(* CODESYS project HomePLC_DIO.library
   Company: Tom Oyen
   Description: Digital in- and outputs
   Version: 1.0
   Placeholder: HomePLC DIO
   Author: Tom Oyen
   Title: HomePLC DIO

Project tree, tasks and I/O mapping:
  libraries: HomePLC Logging, * (Tom Oyen); Tc2_Standard, * (Beckhoff Automation GmbH); Tc2_System, * (Beckhoff Automation GmbH); Tc3_Module, * (Beckhoff Automation GmbH)
  POUs/
    DI/
      DUTs/
        data type E_DICommand
        data type E_DIExecuteSteps
        data type E_DIState
        data type ST_HmiDigitalIn
      function block FB_DigitalIn [ST]: EnableDefer, EnableDoublePress, Execute, SetExternalIn, Command, HmiData, State
      interface I_DigitalIn: EnableDefer, EnableDoublePress, SetExternalIn, Command, HmiData, State
    DO/
      DUTs/
        data type E_DOCommand
        data type E_DOFlashStep
        data type E_DOState
        data type ST_HmiDigitalOut
      function block FB_DigitalOut [ST]: Execute, SetBlinkPeriod, SetCommand, SetFlashTime, BlinkPeriod, Command, FlashTime, HmiData, State
      function block FB_SquareWave [ST]
      interface I_DigitalOut: SetBlinkPeriod, SetCommand, SetFlashTime, BlinkPeriod, Command, FlashTime, HmiData, State
    function block FB_DIO [ST]: Execute, FB_init, Name
    interface I_DIO: Execute, Name
  Project Information/
    function F_GetCompany [ST]
    function F_GetTitle [ST]
    function F_GetVersion [ST]
  Version/
    global variables Global_Version
*)

// POUs/DI/DUTs/E_DICommand
{attribute 'qualified_only'}
{attribute 'strict'}
{attribute 'to_string'}
// Digital input command (generated by digital input)
TYPE E_DICommand :
(
	None		:= 0,		// No input action
	ShortPress	:= 1,		// Input pressed for short amount of time
	LongPress	:= 2,		// Input pressed for longer amount of time but not held
	DoublePress	:= 3,		// Input double pressed
	Hold		:= 4		// Input held for long amount of time
);
END_TYPE

// POUs/DI/DUTs/E_DIExecuteSteps
{attribute 'qualified_only'}
{attribute 'strict'}
// Digital input state machine steps
TYPE E_DIExecuteSteps :
(
	Idle					:= 0,
	FirstShortPressDetected	:= 1,
	WaitForSecondPress		:= 2,
	ShortPressDetected		:= 3,
	DoublePressDetected		:= 4,
	LongPressDetected		:= 5,
	HoldDetected			:= 6,
	WaitUntilReleased		:= 7,
	Reset					:= 8
);
END_TYPE

// POUs/DI/DUTs/E_DIState
{attribute 'qualified_only'}
{attribute 'strict'}
{attribute 'to_string'}
// Digital input state
TYPE E_DIState :
(
	Idle			:= 0,		// No input action
	Pressing1		:= 1,		// Input is being pressed for the first time for a short amount of time
	LongPressing	:= 2,		// Input is being pressed longer
	Pressing2		:= 3,		// Input is being pressed for the second time
	Holding			:= 4,		// Input is being held
	Deferring		:= 5
);
END_TYPE

// POUs/DI/DUTs/ST_HmiDigitalIn
TYPE ST_HmiDigitalIn :
STRUCT
	sName	: STRING;
	eState	: E_DIState;
	bValue	: BOOL;
END_STRUCT
END_TYPE

// POUs/DO/DUTs/E_DOCommand
{attribute 'qualified_only'}
{attribute 'strict'}
{attribute 'to_string'}
// Digital output command (received by digital output)
TYPE E_DOCommand :
(
	None		:= 0,		// No command given
	On			:= 1,		// Turn on
	Off			:= 2,		// Turn off
	Toggle		:= 3,		// Toggle
	Blink		:= 4,		// Blink continuously
	Flash		:= 5		// Flash once (either flash on when already off or flash off when already on)
);
END_TYPE

// POUs/DO/DUTs/E_DOFlashStep
{attribute 'qualified_only'}
{attribute 'strict'}
// Steps when flashing
TYPE E_DOFlashStep :
(
	Start					:= 0,
	ToggleOutput			:= 1,
	WaitForTimer			:= 2,
	RestoreOutput			:= 3,
	End						:= 4
);
END_TYPE

// POUs/DO/DUTs/E_DOState
{attribute 'qualified_only'}
{attribute 'strict'}
{attribute 'to_string'}
// Digital output state
TYPE E_DOState :
(
	Idle			:= 0,		// Idle
	TurnOn			:= 1,		// Turn on
	TurnOff			:= 2,		// Turn off
	Toggle			:= 3,		// Toggle
	Blinking		:= 4,		// Blinking
	Flashing		:= 5		// Flashing	
);
END_TYPE

// POUs/DO/DUTs/ST_HmiDigitalOut
TYPE ST_HmiDigitalOut :
STRUCT
	sName	: STRING;
	eState	: E_DOState;
	bValue	: BOOL;
END_STRUCT
END_TYPE

// Version/Global_Version
{attribute 'TcGenerated'}
{attribute 'no-analysis'}
{attribute 'linkalways'}
// This function has been automatically generated from the project information.
VAR_GLOBAL CONSTANT
	{attribute 'const_non_replaced'}
	stLibVersion_HomePLC_DIO : ST_LibVersion := (iMajor := 1, iMinor := 0, iBuild := 0, iRevision := 0, nFlags := 0, sVersion := '1.0');
END_VAR

// POUs/DI/FB_DigitalIn
// Digital input FB
FUNCTION_BLOCK FB_DigitalIn extends FB_DIO IMPLEMENTS I_DigitalIn
VAR
	ibIn			AT %I*	: BOOL;							// Linked input variable
	bExternalIn				: BOOL;							// External input to trigger this digital input
	eCommand				: E_DICommand;					// Command generated by digital input
	eState					: E_DIState := E_DIState.Idle;	// State of the digital input
	bDoublePressEnabled		: BOOL := FALSE;				// Set to true to enable double press detection
	bDeferEnabled			: BOOL := TRUE;					// Set to true to enable deferring right after input
END_VAR
VAR RETAIN
	nSwitchCount			: UDINT;						// Counter for the number of times the input has switched (0-4294967295)
END_VAR

// Enable/disable deferring right after input
METHOD EnableDefer
VAR_INPUT
	bEnable		: BOOL;		// Set to true to enable deferring right after input
END_VAR
bDeferEnabled := bEnable;
END_METHOD

// Enable/disable double press detection
METHOD EnableDoublePress
VAR_INPUT
	bEnable		: BOOL;		// Set to true to enable double press detection
END_VAR
bDoublePressEnabled := bEnable;
END_METHOD

// Run this method every cycle
METHOD Execute
VAR_INST
	bInput					: BOOL;				// Input obtained from linked digital input or external input
	eStep					: E_DIExecuteSteps;	// State machine state
	fbTimerPressed			: TON;				// Timer to record the time the button was pressed
	fbHoldTimer				: TON;				// Timer to record the time the button was held
	tTimePressed			: TIME;				// Time button was pressed
	fbReleasedTrigger		: F_TRIG;			// Falling edge generated when button is released
	fbWaitSecondPress		: TON;				// Timer to wait for second button press after first press was detected
	fbDeferInput			: TON;				// Timer to defer new input after command
END_VAR
VAR
	sTemp					: STRING;			// Temporary string
END_VAR
// Only run trigger FBs in states where they are used, otherwise an edge may be missed!

// Input = linked digital input or external input
bInput := ibIn OR bExternalIn;

CASE eStep OF
	E_DIExecuteSteps.Idle:
		// Store elapsed time before running FB again
		tTimePressed := fbTimerPressed.ET;
		
		// Set state
		IF bInput THEN
			// State based on time pressed
			IF tTimePressed < T#200MS THEN
				// Pressing first time for short amount of time
				eState := E_DIState.Pressing1;
			ELSIF tTimePressed < T#2000MS THEN
				// Pressing longer but not holding
				eState := E_DIState.LongPressing;
			ELSE
				// Holding
				eState := E_DIState.Holding;
			END_IF
		END_IF
		
		// Run FBs
		fbTimerPressed(IN := bInput, PT := T#2500MS);
		fbHoldTimer(IN := bInput, PT := T#1H);
		fbReleasedTrigger(CLK := bInput);
		
		// When button is released or timer expires
		IF fbReleasedTrigger.Q OR fbTimerPressed.Q THEN			
			// Determine press type based on time pressed
			IF tTimePressed < T#500MS THEN
				// First short press detected
				eStep := E_DIExecuteSteps.FirstShortPressDetected;
			ELSIF tTimePressed < T#2000MS THEN
				// Long press detected
				eStep := E_DIExecuteSteps.LongPressDetected;
			ELSE
				// Hold detected
				// Button is still being held
				eStep := E_DIExecuteSteps.HoldDetected;
			END_IF
		END_IF
		
	E_DIExecuteSteps.FirstShortPressDetected:
		// Reset FB before using it
		fbWaitSecondPress(IN := FALSE);
		
		// Set state
		IF bInput THEN
			// Pressing second time
			eState := E_DIState.Pressing2;
		END_IF
		
		// Check if double press detection is enabled
		IF bDoublePressEnabled THEN
			eStep := E_DIExecuteSteps.WaitForSecondPress;
		ELSE
			eStep := E_DIExecuteSteps.ShortPressDetected;
		END_IF

	E_DIExecuteSteps.WaitForSecondPress:
		// Wait for second press
		
		// Set state
		IF bInput THEN
			// Pressing second time
			eState := E_DIState.Pressing2;
		END_IF
		
		// Run FBs
		fbReleasedTrigger(CLK := bInput);
		fbWaitSecondPress(IN := TRUE, PT := T#200MS);		// Wait x second for second press to occur
		
		// Check button pressed and released again
		IF fbReleasedTrigger.Q THEN
			// Double press detected
			eStep := E_DIExecuteSteps.DoublePressDetected;
		END_IF
		
		// Check if time elapsed, then it was just a single press
		IF fbWaitSecondPress.Q THEN
			// Short press detected
			eStep := E_DIExecuteSteps.ShortPressDetected;
		END_IF
		
	E_DIExecuteSteps.ShortPressDetected:
		// Log
		sTemp := 'Short press ';
		sTemp := CONCAT(sTemp, TIME_TO_STRING(tTimePressed));
		fbLogger.AddDebug(sTemp);
			
		// Set command for one cycle
		eCommand := E_DICommand.ShortPress;
		nSwitchCount := nSwitchCount + 1;
		
		eStep := E_DIExecuteSteps.Reset;
		
	E_DIExecuteSteps.DoublePressDetected:
		// Log
		sTemp := 'Double press ';
		sTemp := CONCAT(sTemp, TIME_TO_STRING(tTimePressed));
		sTemp := CONCAT(sTemp, ' - ');
		sTemp := CONCAT(sTemp, TIME_TO_STRING(fbWaitSecondPress.ET));
		fbLogger.AddDebug(sTemp);
		
		// Set command for one cycle
		eCommand := E_DICommand.DoublePress;
		nSwitchCount := nSwitchCount + 2;
		
		eStep := E_DIExecuteSteps.Reset;
	
	E_DIExecuteSteps.LongPressDetected:
		// Log
		sTemp := 'Long press ';
		sTemp := CONCAT(sTemp, TIME_TO_STRING(tTimePressed));
		fbLogger.AddDebug(sTemp);
		
		// Set command for one cycle
		eCommand := E_DICommand.LongPress;
		nSwitchCount := nSwitchCount + 1;
		
		eStep := E_DIExecuteSteps.Reset;
		
	E_DIExecuteSteps.HoldDetected:
		// Log
		sTemp := 'Hold ';
		sTemp := CONCAT(sTemp, TIME_TO_STRING(tTimePressed));
		fbLogger.AddDebug(sTemp);
		
		// Set command for one cycle
		eCommand := E_DICommand.Hold;
		nSwitchCount := nSwitchCount + 1;
		
		// Hold was detected but button release has not been detected yet
		// Detect button release before returning to idle
		eStep := E_DIExecuteSteps.WaitUntilReleased;
		
	E_DIExecuteSteps.WaitUntilReleased:
		// Reset
		eCommand := E_DICommand.None;
		
		// Store elapsed time before running FB again
		tTimePressed := fbHoldTimer.ET;
		
		// Run FB
		fbHoldTimer(IN := bInput, PT := T#1H);
		fbReleasedTrigger(CLK := bInput);
		
		// Wait until released
		IF fbReleasedTrigger.Q THEN
			// Log
			sTemp := 'Held for ';
			sTemp := CONCAT(sTemp, TIME_TO_STRING(tTimePressed));
			fbLogger.AddDebug(sTemp);
		
			eStep := E_DIExecuteSteps.Reset;
		END_IF
		
	E_DIExecuteSteps.Reset:
		// Reset
		eCommand := E_DICommand.None;
		
		IF bDeferEnabled THEN
			// Deferring enabled
			eState := E_DIState.Deferring;
		
			fbDeferInput(IN := TRUE, PT := T#500MS);
			
			IF fbDeferInput.Q THEN
				fbDeferInput(IN := FALSE);
				eState := E_DIState.Idle;
				eStep := E_DIExecuteSteps.Idle;
			END_IF
		ELSE
			// Reset immediately
			eState := E_DIState.Idle;
			eStep := E_DIExecuteSteps.Idle;
		END_IF
END_CASE
END_METHOD

// Set the external input
METHOD SetExternalIn
VAR_INPUT
	bIn		: BOOL;		// External input value
END_VAR
bExternalIn := bIn;
END_METHOD

// Get the digital input command = translation from on duration of input
PROPERTY Command : E_DICommand
GET
Command := eCommand;
END_GET
END_PROPERTY

// Get HMI data
PROPERTY HmiData : ST_HmiDigitalIn
GET
HmiData.sName := sName;
HmiData.eState := eState;
HmiData.bValue := ibIn or bExternalIn;
END_GET
END_PROPERTY

// Get the digital input state
PROPERTY State : E_DIState
GET
State := eState;
END_GET
END_PROPERTY

END_FUNCTION_BLOCK

// POUs/FB_DIO
// Digital IO abstract FB
{attribute 'reflection'} 
FUNCTION_BLOCK ABSTRACT FB_DIO
VAR
	fbLogger	: class_Tc3EventLogger;			// Logging FB

	// Use attributes to copy instance name to sName
	{attribute 'instance-path'} 
    {attribute 'noinit'} 
    sName		: STRING; 						// Instance name
END_VAR

// Run this method every cycle
METHOD ABSTRACT Execute
END_METHOD

// Perform initialization (implicit call)
METHOD FB_init : BOOL
VAR_INPUT
	bInitRetains : BOOL; // if TRUE, the retain variables are initialized (warm start / cold start)
	bInCopyCode : BOOL;  // if TRUE, the instance afterwards gets moved into the copy code (online change)
END_VAR
// Init logger
fbLogger.Init(sSource := sName, bEnableVerbose := TRUE);
END_METHOD

// Get the name of the IO
PROPERTY Name : STRING
GET
Name := sName;
END_GET
END_PROPERTY

END_FUNCTION_BLOCK

// POUs/DI/I_DigitalIn
// Digital input interface
INTERFACE I_DigitalIn EXTENDS I_DIO

// Enable/disable deferring right after input
METHOD EnableDefer
VAR_INPUT
	bEnable		: BOOL;		// Set to true to enable deferring right after input
END_VAR
END_METHOD

// Enable/disable double press detection
METHOD EnableDoublePress
VAR_INPUT
	bEnable		: BOOL;		// Set to true to enable double press detection
END_VAR
END_METHOD

// Set the external input
METHOD SetExternalIn
VAR_INPUT
	bIn		: BOOL;		// External input value
END_VAR
END_METHOD

// Get the digital input command = translation from on duration of input
PROPERTY Command : E_DICommand
GET
END_GET
END_PROPERTY

// Get HMI data
PROPERTY HmiData : ST_HmiDigitalIn
GET
END_GET
END_PROPERTY

// Get the digital input state
PROPERTY State : E_DIState
GET
END_GET
END_PROPERTY

END_INTERFACE

// POUs/I_DIO
// Interface for digital IO
INTERFACE I_DIO

// Run this method every cycle
METHOD ABSTRACT Execute
END_METHOD

// Get the name of the IO
PROPERTY Name : STRING
GET
END_GET
END_PROPERTY

END_INTERFACE

// POUs/DO/FB_DigitalOut
// Digital output FB
FUNCTION_BLOCK FB_DigitalOut EXTENDS FB_DIO IMPLEMENTS I_DigitalOut
VAR
	obOut		AT %Q*	: BOOL;								// Linked output variable
	eCommand			: E_DOCommand := E_DOCommand.None;	// Command received by digital output
	eState				: E_DOState	:= E_DOState.Idle;		// State of the digital output
	tBlinkPeriod		: TIME := T#2S;						// Square wave period when blinking
	tFlashTime			: TIME := T#2s;						// Time to toggle output when flashing
END_VAR
VAR RETAIN
	nSwitchCount		: UDINT;						// Counter for the number of times the input has switched (0-4294967295)
END_VAR

// Run this method every cycle
METHOD Execute
VAR_INST
	eFlashStep			: E_DOFlashStep;		// Step when flashing
	fbSquareWave		: FB_SquareWave;		// Square wave generator FB
	fbFlashTimer		: TON;					// Flash timer FB
	bOutPrevious		: BOOL;					// Previous output value
	bBlinking			: BOOL;					// True if blinking
END_VAR
// Execute command
CASE eCommand OF
	E_DOCommand.None:	// Do nothing
	E_DOCommand.On:		eState := E_DOState.TurnOn;
	E_DOCommand.Off:	eState := E_DOState.TurnOff;
	E_DOCommand.Toggle:	eState := E_DOState.Toggle;
	E_DOCommand.Blink:	eState := E_DOState.Blinking;
	E_DOCommand.Flash:	eState := E_DOState.Flashing;
END_CASE

// Execute state
CASE eState OF
	E_DOState.Idle:
		// Do nothing
		bBlinking := FALSE;
	
	E_DOState.TurnOn:
		// Turn output on
		IF obOut THEN
			// Already on, nothing to do
		ELSE
			obOut := TRUE;
			
			nSwitchCount := nSwitchCount + 1;
			
			fbLogger.AddDebug(TO_STRING(eCommand));
		END_IF
		
		eState := E_DOState.Idle;
		
	E_DOState.TurnOff:
		// Turn output off
		IF obOut THEN
			obOut := FALSE;
			
			nSwitchCount := nSwitchCount + 1;
			
			fbLogger.AddDebug(TO_STRING(eCommand));
		ELSE
			// Already off, nothing to do
		END_IF
		
		eState := E_DOState.Idle;
		
	E_DOState.Toggle:
		// Toggle output
		obOut := NOT obOut;
		
		nSwitchCount := nSwitchCount + 1;
		
		fbLogger.AddDebug(TO_STRING(eCommand));
		
		eState := E_DOState.Idle;
		
	E_DOState.Blinking:
		// Blink
		fbSquareWave(tPeriod := tBlinkPeriod, bSquareWave => obOut);
		
		IF obOut <> bOutPrevious THEN
			nSwitchCount := nSwitchCount + 1;
		END_IF
		
		bOutPrevious := obOut;
		
		IF eCommand <> E_DOCommand.None AND NOT bBlinking THEN
			fbLogger.AddDebug(TO_STRING(eCommand));
		END_IF
		
		bBlinking := TRUE;
		
	E_DOState.Flashing:
		// Flash once
		CASE eFlashStep OF
			E_DOFlashStep.Start:
				// Reset timer FB
				fbFlashTimer(IN := FALSE);
				
				eFlashStep := E_DOFlashStep.ToggleOutput;
				
			E_DOFlashStep.ToggleOutput:
				// Toggle output
				// Flash = turn on if already off, turn off if already on
				obOut := NOT obOut;
				
				nSwitchCount := nSwitchCount + 1;
				
				eFlashStep := E_DOFlashStep.WaitForTimer;
				
			E_DOFlashStep.WaitForTimer:
				// Wait for timer
				fbFlashTimer(IN := TRUE, PT := tFlashTime);
				
				IF fbFlashTimer.Q THEN
					eFlashStep := E_DOFlashStep.RestoreOutput;
				END_IF
				
			E_DOFlashStep.RestoreOutput:
				// Restore output
				obOut := NOT obOut;
				
				nSwitchCount := nSwitchCount + 1;
				
				eFlashStep := E_DOFlashStep.End;
				
			E_DOFlashStep.End:
				// Reset
				eState := E_DOState.Idle;
				eFlashStep := E_DOFlashStep.Start;
		END_CASE
		
		IF eCommand <> E_DOCommand.None THEN
			fbLogger.AddDebug(TO_STRING(eCommand));
		END_IF
		
END_CASE

// Reset command
eCommand := E_DOCommand.None;
END_METHOD

// Set the square wave period when blinking (default 2s)
METHOD SetBlinkPeriod
VAR_INPUT
	tPeriod		: TIME;			// Blink period
END_VAR
tBlinkPeriod := tPeriod;
END_METHOD

// Set digital output command
METHOD SetCommand
VAR_INPUT
	eCommandIn		: E_DOCommand;	// Command
END_VAR
eCommand := eCommandIn;
END_METHOD

// Set the time to toggle the output when flashing (default 2s)
METHOD SetFlashTime
VAR_INPUT
	tTime		: TIME;			// Flash time
END_VAR
tFlashTime := tTime;
END_METHOD

// Returns the blinking period
PROPERTY BlinkPeriod : TIME
GET
BlinkPeriod := tBlinkPeriod;
END_GET
END_PROPERTY

// Get the command issued to the digital output
PROPERTY Command : E_DOCommand
GET
Command := eCommand;
END_GET
END_PROPERTY

// Returns the flash time
PROPERTY FlashTime : TIME
GET
FlashTime := tFlashTime;
END_GET
END_PROPERTY

// Get HMI data
PROPERTY HmiData : ST_HmiDigitalOut
GET
HmiData.sName := sName;
HmiData.eState := eState;
HmiData.bValue := obOut;
END_GET
END_PROPERTY

// Get the digital output state
PROPERTY State : E_DOState
GET
State := eState;
END_GET
END_PROPERTY

END_FUNCTION_BLOCK

// POUs/DO/I_DigitalOut
// Digital output interface
INTERFACE I_DigitalOut EXTENDS I_DIO

// Set the square wave period when blinking (default 2s)
METHOD SetBlinkPeriod
VAR_INPUT
	tPeriod		: TIME;			// Blink period
END_VAR
END_METHOD

// Set digital output command
METHOD SetCommand
VAR_INPUT
	eCommandIn		: E_DOCommand;		// Command
END_VAR
END_METHOD

// Set the time to toggle the output when flashing (default 2s)
METHOD SetFlashTime
VAR_INPUT
	tTime		: TIME;			// Flash time
END_VAR
END_METHOD

// Returns the blinking period
PROPERTY BlinkPeriod : TIME
GET
END_GET
END_PROPERTY

// Get the command issued to the digital output
PROPERTY Command : E_DOCommand
GET
END_GET
END_PROPERTY

// Returns the flash time
PROPERTY FlashTime : TIME
GET
END_GET
END_PROPERTY

// Get HMI data
PROPERTY HmiData : ST_HmiDigitalOut
GET
END_GET
END_PROPERTY

// Get the digital output state
PROPERTY State : E_DOState
GET
END_GET
END_PROPERTY

END_INTERFACE

// POUs/DO/FB_SquareWave
// Generates a boolean square wave with the given period
FUNCTION_BLOCK FB_SquareWave
VAR_INPUT
	tPeriod			: TIME;			// Period of the square wave
END_VAR
VAR_OUTPUT
	bSquareWave		: BOOL;			// Output square wave
END_VAR
VAR
	fbTimerOn		: TON;			// Timer FB
END_VAR

// Run FB
fbTimerOn();

IF fbTimerOn.Q THEN
	// Timer elapsed
	// Reset timer
	fbTimerOn.IN := FALSE;
	
	// Toggle output
	bSquareWave := NOT bSquareWave;
ELSE
	// Timer running
	// Set period
	fbTimerOn.PT := tPeriod / 2;
	
	// Enable timer
	fbTimerOn.IN := TRUE;	
END_IF

END_FUNCTION_BLOCK

// Project Information/F_GetCompany
// This function has been automatically generated from the project information.
{attribute 'signature_flag' := '1073741824'}
{attribute 'TcGenerated'}
{attribute 'no-analysis'}
FUNCTION F_GetCompany : WSTRING
VAR_INPUT
	
END_VAR

F_GetCompany := "Tom Oyen";

END_FUNCTION

// Project Information/F_GetTitle
// This function has been automatically generated from the project information.
{attribute 'signature_flag' := '1073741824'}
{attribute 'TcGenerated'}
{attribute 'no-analysis'}
FUNCTION F_GetTitle : WSTRING
VAR_INPUT
	
END_VAR

F_GetTitle := "HomePLC DIO";

END_FUNCTION

// Project Information/F_GetVersion
// This function has been automatically generated from the project information.
{attribute 'signature_flag' := '1073741824'}
{attribute 'TcGenerated'}
{attribute 'no-analysis'}
FUNCTION F_GetVersion : ST_LibVersion
VAR_INPUT
	
END_VAR

F_GetVersion.iMajor := 1;
F_GetVersion.iMinor := 0;
F_GetVersion.iBuild := 0;
F_GetVersion.iRevision := 0;
F_GetVersion.sVersion := '1.0';
F_GetVersion.nFlags := 0;

END_FUNCTION
